PROGRAM _Seguridad
VAR
END_VAR

Seguridad.Run := TRUE;
Seguridad.Restart		:= Entradas.ReposicionEmerg OR HMI.Restart;
Seguridad.ErrorAck		:= Entradas.ReposicionEmerg OR HMI.Restart;
Seguridad.ResetPorta	:= Entradas.ReposicionEmerg OR HMI.Restart;

IF HMI.Restart THEN
	HMI.Restart := FALSE;
END_IF

IF NOT Seguridad.PB_Emergencia THEN
	Liquidos.InyectarLiq[1] := FALSE;
	Liquidos.InyectarLiq[2] := FALSE;
	Liquidos.InyectarLiq[3] := FALSE;
	Liquidos.InyectarLiq[4] := FALSE;
	Liquidos.InyectarLiq[5] := FALSE;
	Liquidos.InyectarLiq[6] := FALSE;
	Liquidos.InyectarLiq[7] := FALSE;
	Liquidos.InyectarLiq[8] := FALSE; //a
	Liquidos.InyectarLiq[9] := FALSE;
	Liquidos.InyectarLiq[10] := FALSE;
	Liquidos.InyectarLiq[11] := FALSE;
	Liquidos.InyectarLiq[12] := FALSE;
	Polvos.InyectarPolvo[1] := FALSE;
	Polvos.InyectarPolvo[2] := FALSE;
END_IF

END_PROGRAM

(* stored: Version 1.1.0.1, ProductVersion 3.1.4024.14
   POU _Seguridad: Id {6dd59979-a9f8-4ad0-8d6b-1af8580521a0}, SpecialFunc None *)
